{attribute 'qualified_only'}
{attribute 'strict'}
{attribute 'to_string'}
TYPE enPalletStackerStatus :
(
	Idle := 0,
	Collecting:= 1,
	PinsUitBewegen:= 2,
	LiftBewegen:= 3,
	Omwisselen:= 4,
	Legen:= 5,
	Error:= 6,
	PalletLaden:= 7,
	PinsInBewegen:= 8
);
END_TYPE

(* stored: Version 1.1.0.1
   DUT enPalletStackerStatus: Id {97dcd84d-03a7-492e-b033-c707d2f38cc6} *)
